FUNCTION_BLOCK FB_ModeHome
VAR_INPUT
	bExecute:BOOL;
	bReset: BOOL;
	fVelSet:LREAL:=0;
	fPosSet:LREAL:=0;
	stStatus: ST_AXIS_STATUS;
END_VAR
VAR_OUTPUT
	bError: BOOL;
	nErrorId: UDINT;
	sErrorStr: STRING:=GVL_ErrorCodes.nErrorCodeOKStr;
END_VAR
VAR_IN_OUT
	stCommands: ST_AXIS_COMMAND;
END_VAR
VAR

END_VAR

// Function: Initiate homing of target main  motor
// Actual homing will be performed by the drive.
// Author: Anders Sandström 2018

stCommands.eMotionMode:=e_Motion_mode.ePositioning;
stCommands.bCmd_DriveControlledHoming:=bExecute;
stCommands.fVelocityCommandValue:=GVL_Parameters.fHomeSpeedRpm;
stCommands.fCommandVelocity:=GVL_Parameters.fHomeSpeedRpm;

END_FUNCTION_BLOCK

(* stored: Version 1.1.0.1, ProductVersion 3.1.4024.0
   POU FB_ModeHome: Id {d7b39c30-3a80-4d2f-9742-8a95cc6e84c5}, SpecialFunc None *)
